KUKA KRL program: pickup.src, pickup.dat

--- pickup.src ---
&ACCESS RVP
&REL 22
&PARAM DISKPATH = KRC:\R1\Program\Palletize
DEF  Pickup ( )
   CONTINUE
   PTP BefPikPos C_PTP
   TRIGGER WHEN PATH=-35 DELAY= 0 DO ClsPlt() PRIO=81
   TRIGGER WHEN PATH=-30 DELAY= 0 DO ClsGrp() PRIO=82
   LIN PikPos
   TRIGGER WHEN DISTANCE=0 DELAY=200 DO PusDow() PRIO=83
   LIN AftPikPos C_DIS C_DIS
   PTP EscStpPos C_PTP
   PTP EscBltPos C_PTP
END

DEF PusDow()
$OUT[3]=FALSE
END
DEF ClsGrp()
; Finger
$OUT[1]=FALSE
END
DEF ClsPlt()
; Plate
$OUT[2]=FALSE
END

--- pickup.dat ---
&ACCESS RVP
&REL 22
&PARAM DISKPATH = KRC:\R1\Program\Palletize
DEFDAT  Pickup
;FOLD EXTERNAL DECLARATIONS;%{PE}%MKUKATPBASIS,%CEXT,%VCOMMON,%P
;FOLD GRIPPERTECH EXT
  EXT  H50 (INT:IN, INT:IN ,INT:IN ,GRP_TYP:IN)
;ENDFOLD (GRIPPERTECH EXT)
;FOLD SPOTTECH EXT
  EXT  USERSPOT (S_COMMAND  :IN, SPOT_TYPE:IN)
;ENDFOLD (SPOTTECH EXT)
;FOLD BASISTECH EXT;%{PE}%MKUKATPBASIS,%CEXT,%VEXT,%P
EXT  BAS (BAS_COMMAND  :IN,REAL  :IN )
DECL INT SUCCESS
;ENDFOLD (BASISTECH EXT)
;FOLD USER EXT;%{E}%MKUKATPUSER,%CEXT,%VEXT,%P
;Make here your modifications

;ENDFOLD (USER EXT)
;ENDFOLD (EXTERNAL DECLARATIONS)


DECL E6POS XSTDPICK={X 2176.73755,Y -678.829407,Z -970.623840,A -1.22797132,B 2.32411882E-13,C -180.000,S 2,T 34,E1 0.0,E2 0.0,E3 0.0,E4 0.0,E5 0.0,E6 0.0}
DECL FDAT FStdPick={TOOL_NO 1,BASE_NO 0,IPO_FRAME #BASE,POINT2[] " ",TQ_STATE FALSE}
DECL LDAT LCPDAT1={VEL 2.00000,ACC 100.000,APO_DIST 100.000,APO_FAC 50.0000,AXIS_VEL 100.000,AXIS_ACC 100.000,ORI_TYP #VAR,CIRC_TYP #BASE,JERK_FAC 50.0000,GEAR_JERK 50.0000,EXAX_IGN 0}
DECL E6POS XSTDPICKTOP={X 2176.73755,Y -678.829407,Z -489.025513,A -1.22797120,B -3.74646975E-14,C 180.000,S 2,T 34,E1 0.0,E2 0.0,E3 0.0,E4 0.0,E5 0.0,E6 0.0}
DECL FDAT FStdPickTOP={TOOL_NO 1,BASE_NO 0,IPO_FRAME #BASE,POINT2[] " ",TQ_STATE FALSE}
DECL LDAT LCPDAT6={VEL 2.00000,ACC 100.000,APO_DIST 300.000,APO_FAC 50.0000,AXIS_VEL 100.000,AXIS_ACC 100.000,ORI_TYP #VAR,CIRC_TYP #BASE,JERK_FAC 50.0000,GEAR_JERK 50.0000,EXAX_IGN 0}


ENDDAT
